TYPE ST_CycleData :
STRUCT
//-----------------------------------------------------------------------------------GENERAL------------------------------------------------------------------------------------//	

	bPass				: BOOL;
	bFail				: BOOL;	
	sDate				: STRING;	
	sTime				: STRING;
	
	stHeightTest_CycleData : ST_HeightTest_CycleData;
	stLeakTester_CycleData : ST_LeakTester_CycleData;
	stCamera_CycleData		: ST_Camera_CycleData;


	
	
END_STRUCT
END_TYPE

(* stored: Version 1.1.0.1, ProductVersion 3.1.4024.13
   DUT ST_CycleData: Id {55f28d2e-fb51-4eb3-b909-a265f2991986} *)
